// TIA Portal V20 export
TYPE "typeCmControlNodeSoftCam"
// stored: Namespace Unit1.Em3
   STRUCT
      topTapeAxisX : "Unit1.Em3.typeCmControlNodeSoftCamtopTapeAxisX";
      topTapeAxisY : "Unit1.Em3.typeCmControlNodeSoftCamtopTapeAxisY";
   END_STRUCT;
END_TYPE
